// Brief: Master Arm Standby
FUNCTION_BLOCK PUBLIC FB_StateCtrlStandBy EXTENDS FB_SlaveArmCtrlBase
VAR_INPUT
END_VAR
VAR_OUTPUT
END_VAR
VAR
END_VAR

METHOD PUBLIC init : BOOL
VAR_IN_OUT CONSTANT
	i_slaveArm	:FB_SlaveArm;
END_VAR
VAR_IN_OUT 
	r_slaveArmCtrlCmd :ST_SlaveArmCtrlCmds;
END_VAR
SUPER^.Init(i_slaveArm,r_slaveArmCtrlCmd);

// check if to hold the command joint position unchanged
checkToHoldLastCmds(i_slaveArm,r_slaveArmCtrlCmd);
END_METHOD

END_FUNCTION_BLOCK

(* stored: Version 1.1.0.1, ProductVersion 3.1.4024.12
   POU FB_StateCtrlStandBy: Id {82e389e4-7a38-4619-a14b-0246d1236311}, SpecialFunc None
   Method init: Id {e4eba8ef-1092-44ea-8fed-edb6d236e75a} *)
